{attribute 'linkalways'} 
{attribute 'no_explicit_call' := 'This FB is a CLASS and must be accessed using methods or properties'}
{attribute 'enable_dynamic_creation'}
FUNCTION_BLOCK Node_ContainerType_Vector_USINT EXTENDS Node
VAR
    out : _GUID;
END_VAR

METHOD PUBLIC  Clone : I_Node
VAR
	pNode : POINTER TO Node_ContainerType_Vector_USINT;
END_VAR
pNode := __NEW(Node_ContainerType_Vector_USINT);
Clone := pNode^;
END_METHOD

METHOD FB_init : BOOL
VAR_INPUT
	bInitRetains : BOOL; // if TRUE, the retain variables are initialized (warm start / cold start)
	bInCopyCode : BOOL;  // if TRUE, the instance afterwards gets moved into the copy code (online change)
END_VAR
AddOutput('out', out);
END_METHOD

METHOD PROTECTED OnExecute
out.Value := ContainerType_Vector_USINT;
END_METHOD

END_FUNCTION_BLOCK

(* stored: Version 1.1.0.1, ProductVersion 3.1.4026.17
   POU Node_ContainerType_Vector_USINT: Id {ff0e9d1d-faf4-01ca-143e-7c0f2427ddb0}, SpecialFunc None
   Folder Constructor: Id {beba9eac-d8a7-08e8-28d9-fdfef3adceb0}
   Method Clone: Id {682ba460-8064-036d-0a16-2af9fb954e6e}
   Method FB_init: Id {88e465f4-3be4-0b35-0f07-43b99ce0a435}
   Method OnExecute: Id {515776f1-4445-0748-156c-364e88dc5efe} *)
